# EPICS autosave request: iocBoot/iocpmcvtest/auto_settings.req
file motor_settings.req P=MLL:,M=pmcv1
file motor_settings.req P=MLL:,M=pmcv2
file motor_settings.req P=MLL:,M=pmcv3
